// TIA Portal V16 export
// export: Created 2024-09-05T17:40:14.9389441Z, ExportSetting WithDefaults, DisplayName Totally Integrated Automation Portal, DisplayVersion V16 Update 6, DisplayName TIA Portal Version Control Interface, DisplayVersion V16 Update 2, DisplayName TIA Portal Openness, DisplayVersion V16 Update 6, DisplayName STEP 7 Professional, DisplayVersion V16 Update 6, DisplayName STEP 7 Safety, DisplayVersion V16, DisplayName WinCC Advanced, DisplayVersion V16 Update 6
TYPE "UDT_SafetyLevels"
// stored: IsFailsafeCompliant false
   STRUCT
      "Level_1L+" : Bool;
      "Level_2L+" : Bool;
      "Level_3L+" : Bool;
      "Level_4L+" : Bool;
      "Level_5L+" : Bool;
      "Level_6L+" : Bool;
      "Level_7L+" : Bool;
      "Level_8L+" : Bool;
      "Level_9L+" : Bool;
      "Level_10L+" : Bool;
      SystemReady : Bool;
   END_STRUCT;
END_TYPE
